(*
    TcXunit interpreter fixture (TcXunit-w5x.8). TcUnit-style suite exercising
    the interpreter's native-stub TEST()/TEST_FINISHED()/AssertTrue/
    AssertEquals_INT surface (TcXunit-w5x.7) against FB_Counter and
    FB_ClampedCounter.
*)
FUNCTION_BLOCK FB_CounterTests EXTENDS TcUnit.FB_TestSuite

CounterStartsAtZero();
IncrementAddsDelta();
DecrementClampsAtZero();
ClampedCounterIncrementRespectsCeiling();

METHOD PRIVATE CounterStartsAtZero
VAR
	counter : FB_Counter;
END_VAR
TEST('CounterStartsAtZero');

AssertEquals_INT(Expected := 0,
                  Actual := counter.GetValue(),
                  Message := 'fresh counter');

TEST_FINISHED();
END_METHOD

METHOD PRIVATE IncrementAddsDelta
VAR
	counter : FB_Counter;
END_VAR
TEST('IncrementAddsDelta');

counter.Increment(delta := 3);

AssertEquals_INT(Expected := 3,
                  Actual := counter.GetValue(),
                  Message := 'after Increment(3)');

TEST_FINISHED();
END_METHOD

METHOD PRIVATE DecrementClampsAtZero
VAR
	counter : FB_Counter;
END_VAR
TEST('DecrementClampsAtZero');

counter.Decrement(delta := 5);

AssertEquals_INT(Expected := 0,
                  Actual := counter.GetValue(),
                  Message := 'Decrement below zero');

TEST_FINISHED();
END_METHOD

METHOD PRIVATE ClampedCounterIncrementRespectsCeiling
VAR
	counter : FB_ClampedCounter;
END_VAR
TEST('ClampedCounterIncrementRespectsCeiling');

counter.Increment(delta := 999);

AssertTrue(Condition := (counter.GetValue() = 10),
           Message := 'Increment did not clamp at ceiling');

TEST_FINISHED();
END_METHOD

END_FUNCTION_BLOCK

(* stored: Version 1.1.0.1, ProductVersion 3.1.4026.18
   POU FB_CounterTests: Id {a1b2c3d4-0003-4a1a-8b1b-000000000001}, SpecialFunc None
   Method CounterStartsAtZero: Id {a1b2c3d4-0003-4a1a-8b1b-000000000002}
   Method IncrementAddsDelta: Id {a1b2c3d4-0003-4a1a-8b1b-000000000003}
   Method DecrementClampsAtZero: Id {a1b2c3d4-0003-4a1a-8b1b-000000000004}
   Method ClampedCounterIncrementRespectsCeiling: Id {a1b2c3d4-0003-4a1a-8b1b-000000000005} *)
